(*
	Log Error message to TwinCAT console
*)
{attribute 'hide_all_locals'}
FUNCTION F_LogError : BOOL
VAR_INPUT
	sMessage : T_MAXSTRING;
END_VAR

VAR CONSTANT	
	LOGHEADER		: T_MAXSTRING := 'Open Commissioning: %s';
END_VAR

ADSLOGSTR(ADSLOG_MSGTYPE_ERROR, LOGHEADER, sMessage);

END_FUNCTION

(* stored: Version 1.1.0.1, ProductVersion 3.1.4024.12
   POU F_LogError: Id {4f6bc53c-00e9-0ffe-0447-891bfa4a8ab9}, SpecialFunc None *)
